(* CoDeSys 2.3.9.31 project: test1.pro *)
(* Title: Maschine *)
(* Author: Beckhoff Industrie Elektronic *)
(* Description: Sample from the Manual
'TwinCAT - first Steps' *)
(* Libraries: Standard.lib 5.6.98 11:03:02 *)

(* Task configuration *)
TASK Standard (PRIORITY := 0, INTERVAL := T#10ms);
	MAIN
END_TASK

(* Global variable list: Globale_Variablen *)
VAR_GLOBAL
	engine		AT %QX0.0:	BOOL;
	deviceUp	AT %QX0.1:	BOOL;
	deviceDown	AT %QX0.2:	BOOL;
	timerUp:					TON;
	timerDown:				TON;
	steps:					BYTE;
	count:					UINT := 0;
	devSpeed:				TIME := t#10ms;
	devTimer:				TON;
	switch: BOOL;
END_VAR

(* POU MAIN, ST *)
PROGRAM MAIN
VAR
	IN_BTN_1: BOOL;
	IN_BTN_2: BOOL;

	IN_MBW_1: BOOL;
	IN_MBW_2: BOOL;
	IN_MBW_3: BOOL;

	OUT_LMP_1:BOOL;
	OUT_LMP_2:BOOL;
	OUT_LMP_3:BOOL;

	OUT_LMP_1_CTL:FB_SON_SOFF_MODBUS;
	OUT_LMP_2_CTL:FB_LON_LOFF_MODBUS;
	OUT_LMP_3_CTL:FB_LON_SOFF_MODBUS;

	MB1:R_TRIG;
END_VAR
MB1(CLK:=IN_MBW_3);

OUT_LMP_1_CTL(IN:=IN_BTN_1, IN_MB:=IN_MBW_1,  TC:=t#1000ms);
OUT_LMP_2_CTL(IN:=IN_BTN_1, IN_MB:=IN_MBW_2,  TC:=t#1000ms);
OUT_LMP_3_CTL(IN:=IN_BTN_2, IN_MB:=MB1.Q,  TC:=t#1000ms);

OUT_LMP_1 := OUT_LMP_1_CTL.Q;
OUT_LMP_2 := OUT_LMP_2_CTL.Q;
OUT_LMP_3 := OUT_LMP_3_CTL.Q;
END_PROGRAM

(* POU FB_SON_SOFF_MODBUS, ST *)
FUNCTION_BLOCK FB_SON_SOFF_MODBUS
VAR_INPUT
	IN:BOOL;
	IN_MB:BOOL;
	TC:TIME;
END_VAR
VAR_OUTPUT
	Q:BOOL := FALSE;
END_VAR
VAR
	MEM:BOOL := FALSE;
	TX:TP;
	FLAG:BOOL := FALSE;
END_VAR
TX(IN := IN, PT := TC);
IF IN THEN
	FLAG:=TRUE;
ELSIF NOT IN AND FLAG THEN
	FLAG := FALSE;
	IF TX.Q THEN
		Q := NOT Q;
	END_IF
END_IF

IF IN_MB THEN
	Q := NOT Q;
END_IF

MEM := Q;
END_FUNCTION_BLOCK

(* POU FB_LON_LOFF_MODBUS, ST *)
FUNCTION_BLOCK FB_LON_LOFF_MODBUS
VAR_INPUT
	IN:BOOL;
	IN_MB:BOOL;
	TC:TIME;
END_VAR
VAR_OUTPUT
	Q:BOOL := FALSE;
END_VAR
VAR
	TX:TON;
	MEM:BOOL := FALSE;
END_VAR
TX(IN := IN, PT := TC);

IF IN AND TX.Q AND NOT MEM THEN
	Q := NOT Q;
END_IF

IF IN_MB THEN
	Q := NOT Q;
END_IF

MEM := TX.Q;
END_FUNCTION_BLOCK

(* POU FB_LON_SOFF_MODBUS, ST *)
FUNCTION_BLOCK FB_LON_SOFF_MODBUS
VAR_INPUT
	IN:BOOL;
	IN_MB:BOOL;
	TC:TIME;
END_VAR
VAR_OUTPUT
	Q:BOOL := FALSE;
END_VAR
VAR
	TX:TON;
	MEM:BOOL := FALSE;
	MEM2:BOOL := FALSE;
END_VAR
TX(IN := IN, PT := TC);

IF IN AND NOT MEM THEN
	IF NOT Q AND TX.Q THEN
		Q := NOT Q;
	ELSIF Q THEN
		Q := NOT Q;
	END_IF
END_IF

IF IN_MB THEN
	Q := NOT Q;
END_IF

MEM := TX.Q;
END_FUNCTION_BLOCK

(* POU FB_SON_LOFF_MODBUS, ST *)
FUNCTION_BLOCK FB_SON_LOFF_MODBUS
VAR_INPUT
	IN:BOOL;
	IN_MB:BOOL;
	TC:TIME;
END_VAR
VAR_OUTPUT
	Q:BOOL := FALSE;
END_VAR
VAR
	TX:TON;
	MEM:BOOL := FALSE;
END_VAR
TX(IN := IN, PT := TC);

IF IN AND NOT MEM THEN
	IF Q AND TX.Q  THEN
		Q := NOT Q;
	ELSIF NOT Q THEN
		Q := NOT Q;
	END_IF
END_IF

IF IN_MB THEN
	Q := NOT Q;
END_IF

MEM := TX.Q;
END_FUNCTION_BLOCK

(* POU FB_SON_SOFF_MODBUS_SINGLE, ST *)
FUNCTION_BLOCK FB_SON_SOFF_MODBUS_SINGLE
VAR_INPUT
	IN:BOOL;
	IN_MB:BOOL;
END_VAR
VAR_OUTPUT
	Q:BOOL := FALSE;
END_VAR
VAR
	MEM:BOOL := FALSE;
	CTL:BOOL;
END_VAR
CTL:=IN OR IN_MB;
IF CTL AND NOT MEM THEN
   Q:= NOT Q;
END_IF

MEM := CTL;
END_FUNCTION_BLOCK

(* Visualisation MAIN
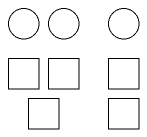
ellipse at (10,10)-(41,41): alarm colour if MAIN.OUT_LMP_1
rectangle at (30,100)-(61,131): alarm colour if MAIN.IN_BTN_1; taps MAIN.IN_BTN_1
ellipse at (50,10)-(81,41): alarm colour if MAIN.OUT_LMP_2
rounded rectangle at (10,60)-(41,91): alarm colour if MAIN.IN_MBW_1; taps MAIN.IN_MBW_1
rounded rectangle at (50,60)-(81,91): alarm colour if MAIN.IN_MBW_2; taps MAIN.IN_MBW_2
rectangle at (110,100)-(141,131): alarm colour if MAIN.IN_BTN_2; taps MAIN.IN_BTN_2
ellipse at (110,10)-(141,41): alarm colour if MAIN.OUT_LMP_3
rounded rectangle at (110,60)-(141,91): alarm colour if MAIN.IN_MBW_3; taps MAIN.IN_MBW_3
*)
